// LS Electric XG5000 project: 타이머
// PLC NewPLC

PROGRAM NewProgram (task: 스캔 프로그램)

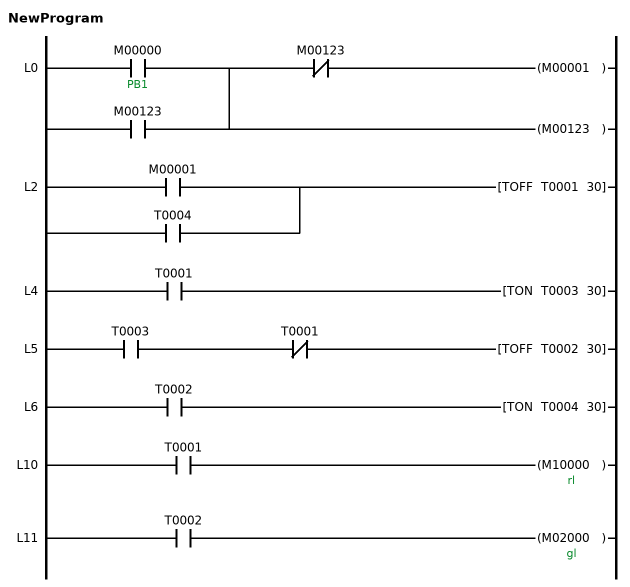
; L0
LOAD      M00000	// PB1
OR        M00123
MPUSH
AND NOT   M00123
OUT       M00001
MPOP
OUT       M00123
; L2
LOAD      M00001
OR        T0004
TOFF      T0001 30
; L4
LOAD      T0001
TON       T0003 30
; L5
LOAD      T0003
AND NOT   T0001
TOFF      T0002 30
; L6
LOAD      T0002
TON       T0004 30
; L10
LOAD      T0001
OUT       M10000	// rl
; L11
LOAD      T0002
OUT       M02000	// gl